INTERFACE I_XTS

METHOD DisableXTS : BOOL
VAR_INPUT
END_VAR
END_METHOD

METHOD EnableXTS : BOOL
VAR_INPUT
END_VAR
END_METHOD

METHOD IsInitialised : BOOL
END_METHOD

METHOD IsXtsIdle : BOOL
VAR_INPUT
END_VAR
END_METHOD

METHOD IsXtsReady : BOOL
VAR_INPUT
END_VAR
END_METHOD

METHOD PUBLIC Abstract MoverHomeSequence : BOOL
VAR_INPUT
END_VAR
END_METHOD

METHOD RegisterMovers : HRESULT
VAR_INPUT
	MyMover : I_XtsMover;
END_VAR
END_METHOD

METHOD StopXts : BOOL
VAR_INPUT
END_VAR
END_METHOD

END_INTERFACE

(* stored: Version 1.1.0.1
   Itf I_XTS: Id {eb22a7d8-6cc9-41fe-bacb-ecb9c288212d}
   Method DisableXTS: Id {d730e6bc-30f4-400f-83c5-0a8ef7530dc6}
   Method EnableXTS: Id {a90bf243-5fbb-42eb-a2e5-eb1ea9f490a9}
   Method IsInitialised: Id {e1565fab-ac95-48ac-ae78-e46b6110b4fc}
   Method IsXtsIdle: Id {a58467b2-fd55-49b7-9538-35b2ad34103b}
   Method IsXtsReady: Id {88e988d8-b3fd-4023-a27f-e2263614dcbf}
   Method MoverHomeSequence: Id {ac0ec977-8522-4017-9641-ad2a4c242c82}
   Method RegisterMovers: Id {e65bc655-b1b5-4ed3-91eb-2d51871a4d75}
   Method StopXts: Id {d7591d56-8a8c-46a1-bfd3-85f1f168760d} *)
